(* PLC project  *)

CONFIGURATION Empty_Module_4
END_CONFIGURATION
